(* IEC 61131-3 sources: IR_12059_group_03/labs/lab_01/build/OpenPLC Runtime v4/src, 1 file *)

(* ---- program.st ---- *)
PROGRAM main
  VAR
    BUTTON AT %QX0.0 : BOOL;
    MOTOR AT %QX0.1 : BOOL;
  END_VAR

  MOTOR := BUTTON;
END_PROGRAM

CONFIGURATION Config0

  RESOURCE Res0 ON PLC
    TASK task0(INTERVAL := T#20ms,PRIORITY := 1);
    PROGRAM instance0 WITH task0 : main;
  END_RESOURCE
END_CONFIGURATION
